FUNCTION_BLOCK FB_Animal
VAR
    sOutput : STRING := '';
END_VAR

METHOD M_Eat : BOOL
VAR_INPUT
END_VAR
THIS^.sOutput := 'Animal eats food';
END_METHOD

END_FUNCTION_BLOCK

(* stored: Version 1.1.0.1, ProductVersion 3.1.4024.16
   POU FB_Animal: Id {75d990de-4ce1-4c07-8dcb-89fbf4624ec9}, SpecialFunc None
   Method M_Eat: Id {adae790b-d64c-401e-879b-efb52f712bc3} *)
